// TIA Portal project "Fill_Tank_S7-1200_V14" (V14)
// Vorlageprojekt für das Buch mit Zielsystem S7-1200

(* hardware
DEVICE "S7-1200-Station_1"  S7-1200 Station
   slot 0: "Baugruppenträger_0"  Rack  V1.0
   slot 1: "PLC_1"  CPU 1214C DC/DC/DC  6ES7 214-1AG40-0XB0  V4.2
*)

// ===== PLC "PLC_1"  CPU 1214C DC/DC/DC =====

VAR_GLOBAL   // PLC tag table "Standard-Variablentabelle"
   "En_Fill_Timer" AT %M0.0 : Bool;   // Enable fill tank timer
   "Filling_current_time" AT %MD30 : Time;
   "En_Discharge_Timer" AT %M0.1 : Bool;
   "Discharging_current_time" AT %MD31 : Time;
   "Filling_Time_sec" AT %QW30 : Word;
END_VAR

VAR_GLOBAL   // PLC tag table "Tank_Tags"
   "FIO_Running" AT %I0.0 : Bool;
   "Fill" AT %I0.1 : Bool;
   "Discharge" AT %I0.2 : Bool;
   "Fill_Valve" AT %Q0.0 : Bool;
   "Filling_Light" AT %Q0.1 : Bool;
   "Discharge_Valve" AT %Q0.2 : Bool;
   "Discharging_Light" AT %Q0.3 : Bool;
END_VAR

// folder: System blocks/Program resources

DATA_BLOCK "Fill_Tank_Timer"   // DB1
{ S7_Optimized_Access := 'TRUE' }
AUTHOR : Simatic
FAMILY : IEC
NAME : IEC_TMR
VERSION : 1.0
// stored: InstanceOfName IEC_TIMER
"IEC_TIMER"
BEGIN
END_DATA_BLOCK

DATA_BLOCK "Discharge_Tank_Timer"   // DB2
{ S7_Optimized_Access := 'TRUE' }
AUTHOR : Simatic
FAMILY : IEC
NAME : IEC_TMR
VERSION : 1.0
// stored: InstanceOfName IEC_TIMER
"IEC_TIMER"
BEGIN
END_DATA_BLOCK

// folder: (top level)

FUNCTION "Tank" : Void   // FC1, LAD
{ S7_Optimized_Access := 'TRUE' }
VERSION : 0.1
   VAR_TEMP
      Filling_Time : DInt;
      K_MUX_SLECTOR : Bool;
   END_VAR
BEGIN

REGION Network 1: Enable fill tank timer
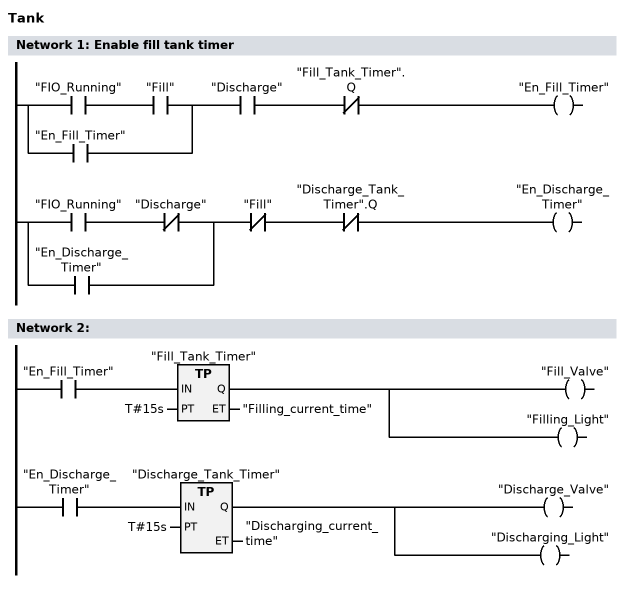
   RUNG wire#powerrail
      Contact( "FIO_Running" )
      Contact( "Fill" )
      wire#w1
      Contact( "Discharge" )
      I_Contact( "Fill_Tank_Timer".Q )
      Coil( "En_Fill_Timer" )
   END_RUNG
   RUNG wire#powerrail
      Contact( "En_Fill_Timer" )
   END_RUNG wire#w1
   RUNG wire#powerrail
      Contact( "FIO_Running" )
      I_Contact( "Discharge" )
      wire#w2
      I_Contact( "Fill" )
      I_Contact( "Discharge_Tank_Timer".Q )
      Coil( "En_Discharge_Timer" )
   END_RUNG
   RUNG wire#powerrail
      Contact( "En_Discharge_Timer" )
   END_RUNG wire#w2
   // the same network as SCL:
   "En_Fill_Timer" := (("FIO_Running" AND "Fill") OR "En_Fill_Timer") AND "Discharge" AND NOT "Fill_Tank_Timer".Q;
   "En_Discharge_Timer" := (("FIO_Running" AND NOT "Discharge") OR "En_Discharge_Timer") AND NOT "Fill" AND NOT "Discharge_Tank_Timer".Q;
END_REGION

REGION Network 2
   "Fill_Tank_Timer".TP(IN := "En_Fill_Timer", PT := T#15s, ET => "Filling_current_time");
   "Fill_Valve" := "Fill_Tank_Timer".Q;
   "Filling_Light" := "Fill_Tank_Timer".Q;
   "Discharge_Tank_Timer".TP(IN := "En_Discharge_Timer", PT := T#15s, ET => "Discharging_current_time");
   "Discharge_Valve" := "Discharge_Tank_Timer".Q;
   "Discharging_Light" := "Discharge_Tank_Timer".Q;
END_REGION
END_FUNCTION

FUNCTION "MHJ-PLC-Lab-Function-S71200" : Void   // FC9000, SCL
{ S7_Optimized_Access := 'TRUE' }
VERSION : 0.1
   VAR_TEMP
      rdTimeReturn : Int;
      outputTime : DTL;
      SyncVal : Byte;
      forVal : Int;
      forVal_2 : Int;
      Value : Byte;
   END_VAR
   VAR CONSTANT
      CompVal : Byte := 16#34;
      Value_01 : Byte := 16#11;
      Value_01_DW : DWord := 16#A165_D992;
      Value_02_DW : DWord := 16#58BE_4401;
   END_VAR
BEGIN

   #Value:=PEEK(area := 16#82,
        dbNumber := 0,
        byteOffset := 511);
   #Value := #Value + 1;

   POKE(area := 16#82,
        dbNumber := 0,
        byteOffset := 511,
        value := #Value);

   POKE(area:=16#81,
        dbNumber:=0,
        byteOffset:=1016,
        value:=#Value_01_DW);
   POKE(area := 16#81,
        dbNumber := 0,
        byteOffset := 1020,
        value := #Value_02_DW);

   POKE(area := 16#81,
        dbNumber := 0,
        byteOffset := 511,
        value := B#16#00);

   FOR #forVal := 0 TO 120 DO
       FOR #forVal_2:=0 TO 10 DO
           #rdTimeReturn:=RD_SYS_T(#outputTime);
           #rdTimeReturn := WR_SYS_T(#outputTime);
           #rdTimeReturn := RD_SYS_T(#outputTime);
           #rdTimeReturn := WR_SYS_T(#outputTime);
       END_FOR;
       #SyncVal:= PEEK(area := 16#81,
                      dbNumber := 0,
                      byteOffset := 511);
       IF #SyncVal = #CompVal THEN
          GOTO M_1;
       END_IF;
   END_FOR;
   RETURN;

   M_1:
   POKE(area := 16#81,
        dbNumber := 0,
        byteOffset := 511,
        value := B#16#0);
END_FUNCTION

ORGANIZATION_BLOCK "Main"   // OB1, FBD, ProgramCycle
TITLE = "Main Program Sweep (Cycle)"
{ S7_Optimized_Access := 'TRUE' }
VERSION : 0.1
   VAR_INPUT
      Initial_Call : Bool;   // Initial call of this OB
      Remanence : Bool;   // =True, if remanent data are available
   END_VAR
BEGIN

REGION Network 1: Konnektierungsbaustein für PLC-Lab
   // Im Netzwerk 1 wird der Konnektierungsbaustein für PLC-Lab aufgerufen.
   // Dieser Aufruf darf nicht entfernt werden!
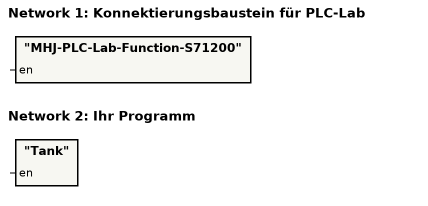
   "MHJ-PLC-Lab-Function-S71200"();
END_REGION

REGION Network 2: Ihr Programm
   // Schreiben Sie ab Netzwerk 2 Ihr Programm
   "Tank"();
END_REGION
END_ORGANIZATION_BLOCK